GLOBALCONSTANTS DefaultPool_AI (* Global constants *)
  PACKAGE Uebungen::const::UT::AI;
  VAR_GLOBAL CONSTANT
    WorkingSet : UINT := 0;
    DataMask_M1 : UINT := 1000;
    DataMask_AI1 : UINT := 1001;
    DataMask_AI2 : UINT := 1002;
    DataMask_AI3 : UINT := 1003;
    DataMask_AI4 : UINT := 1004;
    Container_Q : UINT := 3000;
    SoftKeyMask_AI : UINT := 4000;
    SoftKey_Ausgaenge : UINT := 5000;
    SoftKey_AI1 : UINT := 5001;
    SoftKey_AI2 : UINT := 5002;
    SoftKey_AI3 : UINT := 5003;
    SoftKey_AI4 : UINT := 5004;
    Button_Q01 : UINT := 6001;
    Button_Q02 : UINT := 6002;
    Button_Q03 : UINT := 6003;
    Button_Q04 : UINT := 6004;
    Button_Q05 : UINT := 6005;
    Button_Q06 : UINT := 6006;
    Button_Q07 : UINT := 6007;
    Button_Q08 : UINT := 6008;
    Button_Q09 : UINT := 6009;
    Button_Q10 : UINT := 6010;
    Button_Q11 : UINT := 6011;
    Button_Q12 : UINT := 6012;
    NumberVariable_AI_I01 : UINT := 21000;
    NumberVariable_AI_I02 : UINT := 21001;
    NumberVariable_AI_I03 : UINT := 21002;
    NumberVariable_AI_I04 : UINT := 21003;
    NumberVariable_AI_I05 : UINT := 21004;
    NumberVariable_AI_I06 : UINT := 21005;
    NumberVariable_AI_I07 : UINT := 21006;
    NumberVariable_AI_I08 : UINT := 21007;
    OutputNumber_Tick : UINT := 12020;
    FontAttributes_6x8 : UINT := 23000;
    FontAttributes_24x32 : UINT := 23001;
    FontAttributes_16x16 : UINT := 23002;
    Logos_icon : UINT := 20500;
    AuxFunction2_X1 : UINT := 31000;
  END_VAR
END_GLOBALCONSTANTS
